PROGRAM Axis03_Interlock
VAR
	Always_ON	:	BOOL	:=TRUE	;//상시 ON 
	Always_OFF	:	BOOL	:=FALSE	;//상시 OFF
END_VAR

// NETWORK 1

END_PROGRAM

(* stored: Version 1.1.0.1, ProductVersion 3.1.4024.15
   POU Axis03_Interlock: Id {55902515-fa66-4c8c-b0c4-11bac34c4f15}, SpecialFunc None *)
